TYPE "AreaInterface"
VERSION : 0.1
// Block: AreaInterface
   STRUCT
      EStop : Bool;
      Man : Bool;
      Aut : Bool;
      Cycle : Bool;
      StopInPhase : Bool;
      StopProgrammed : Bool;
      RstAlarms : Bool;
      ManOneShot : Bool;
      AutOneShot : Bool;
      CycleOneShot : Bool;
      CheckAutReady : Bool;
   END_STRUCT;

END_TYPE
